TYPE "LBP_typeModeGroup"
TITLE = Mode group signals / Señales de grupo de modos de operación / Betriebsartengruppe Signale
// User data type for block LBP_ModeGroup [DB11] / Tipo de dato de usuario para bloque LBP_ModeGroup [DB11] / Anwender-Datentyp für Baustein LBP_ModeGroup [DB11]
// stored: IsFailsafeCompliant false
   STRUCT
      A_AUTO : Bool;   // Betriebsart AUTOMATIC / Operating mode AUTOMATIC / Modo de operación AUTOMÁTICO
      A_MDA : Bool;   // Betriebsart MDA / Operating mode MDA / Modo de operación MDA
      A_JOG : Bool;   // Betriebsart JOG / Operating mode JOG / Modo de operación JOG
      f0_3 : Bool;
      A_MCDisable : Bool;   // Betriebsartenwechsel deaktivieren / Mode change disable / Desactivar cambio de modo de operación
      A_MGStop : Bool;   // Betriebsartengruppe Stopp / Mode group stop / Parada de grupo de modos de operación
      A_MGStopASp : Bool;   // Betriebsartengruppe Stopp Achsen plus Spindel / Mode group stop axes plus spindle / Parada de grupo de modos de operación ejes y cabezal
      A_MGReset : Bool;   // Betriebsartengruppe Reset / Mode group reset / Reset de grupo de modos de operación
      A_TEACHIN : Bool;   // Maschinenfunktion TEACH IN / Machine function TEACH IN / Función de máquina TEACH IN
      A_REPOS : Bool;   // Maschinenfunktion REPOS / Machine function REPOS / Función de máquina REPOS
      A_REF : Bool;   // Maschinenfunktion REF / Machine function REF / Función de máquina REF
      f1_3 : Bool;
      f1_4 : Bool;
      f1_5 : Bool;
      A_SingleBlock_B : Bool;   // Einzelsatz Typ B / Single block type B / Secuencia individual tipo B
      A_SingleBlock_A : Bool;   // Einzelsatz Typ A / Single block type A / Secuencia individual tipo A
      A_INC1 : Bool;   // INC1
      A_INC10 : Bool;   // INC10
      A_INC100 : Bool;   // INC100
      A_INC1000 : Bool;   // INC1000
      A_INC10000 : Bool;   // INC10000
      A_INCVar : Bool;   // INC-Variable / INC variable / Variable INC
      A_ContManTravel : Bool;   // Kontinuierliches Verfahren von Hand / Continuous manual travel / Desplazamiento continuo a mano
      f2_7 : Bool;
      f3 : Byte;
      E_MMC_AUTO : Bool;   // HMI Betriebsart Strobe AUTOMATIC / HMI mode strobe AUTOMATIC / Modo de operación HMI strobe AUTOMÁTICO
      E_MMC_MDA : Bool;   // HMI Betriebsart Strobe MDA / HMI mode strobe MDA / Modo de operación HMI strobe MDA
      E_MMC_JOG : Bool;   // HMI Betriebsart Strobe JOG / HMI mode strobe JOG / Modo de operación HMI strobe JOG
      f4_3 : Bool;
      f4_4 : Bool;
      f4_5 : Bool;
      f4_6 : Bool;
      f4_7 : Bool;
      E_MMC_TEACHIN : Bool;   // HMI Maschinenfunktion Strobe TEACH IN / HMI machine function strobe TEACH IN / Función de máquina HMI strobe TEACH IN
      E_MMC_REPOS : Bool;   // HMI Maschinenfunktion Strobe REPOS / HMI machine function strobe REPOS / Función de máquina HMI strobe REPOS
      E_MMC_REF : Bool;   // HMI Maschinenfunktion Strobe REF / HMI machine function strobe REF / Función de máquina HMI strobe REF
      f5_3 : Bool;
      f5_4 : Bool;
      f5_5 : Bool;
      f5_6 : Bool;
      f5_7 : Bool;
      E_AUTO : Bool;   // Aktive Betriebsart AUTOMATIC / Active operating mode AUTOMATIC / Modo de operación activo AUTOMÁTICO
      E_MDA : Bool;   // Aktive Betriebsart MDA / Active operating mode MDA / Modo de operación activo MDA
      E_JOG : Bool;   // Aktive Betriebsart JOG / Active operating mode JOG / Modo de operación activo JOG
      E_MGOK : Bool;   // Betriebsartengruppe bereit / Mode group ready / Grupo de modos de operación listo
      E_MGreseted : Bool;   // Betriebsartengruppe Reset durchgeführt / Mode group reset performed / Reset de grupo de modos de operación realizado
      E_NCKintJOG : Bool;   // NCK interner JOG aktiv / NCK internal JOG active / NCK JOG interno activo
      f6_6 : Bool;
      E_ChanReset : Bool;   // Alle Kanäle in Reset-Mode / All channels in reset state / Todos los canales en modo Reset
      E_TEACHIN : Bool;   // Aktive Maschinenfunktion TEACH IN / Active machine function TEACH IN / Función de máquina activa TEACH IN
      E_REPOS : Bool;   // Aktive Maschinenfunktion REPOS / Active machine function REPOS / Función de máquina activa REPOS
      E_REF : Bool;   // Aktive Maschinenfunktion REF / Active machine function REF / Función de máquina activa REF
      f7_3 : Bool;
      f7_4 : Bool;
      f7_5 : Bool;
      f7_6 : Bool;
      f7_7 : Bool;
      E_INC1 : Bool;   // INC1
      E_INC10 : Bool;   // INC10
      E_INC100 : Bool;   // INC100
      E_INC1000 : Bool;   // INC1000
      E_INC10000 : Bool;   // INC10000
      E_INCVar : Bool;   // INC-Variable / INC variable / Variable INC
      E_ContManTravelAct : Bool;   // Kontinuierliches manuelles Verfahren aktiv / Continuous manual travel active / Desplazamiento manual continuo activo
      f8_7 : Bool;
      f9 : Byte;
      E_HMI_INC1 : Bool;   // INC1 vom HMI / INC1 from HMI / INC1 de HMI
      E_HMI_INC10 : Bool;   // INC10 vom HMI / INC10 from HMI / INC10 de HMI
      E_HMI_INC100 : Bool;   // INC100 vom HMI / INC100 from HMI / INC100 de HMI
      E_HMI_INC1000 : Bool;   // INC1000 vom HMI / INC1000 from HMI / INC1000 de HMI
      E_HMI_INC10000 : Bool;   // INC10000 vom HMI / INC10000 from HMI / INC10000 de HMI
      E_HMI_INCVar : Bool;   // INC-Variable vom HMI / INC variable from HMI / Variable INC de HMI
      E_HMI_ContManTravel : Bool;   // Kontinuierliches manuelles Verfahren vom HMI aktiv / Continuous manual travel active from HMI / Desplazamiento manual continuo activo desde HMI
      f10_7 : Bool;
      f11 : Byte;
      f12 : Array[12..19] of Byte;
      MG : Array[2..10] of Struct   // Nächste Betriebsartengruppe vom DBB20, wie bisher / next mode group from DBB20, as before / Próximo grupo de modos de operación del DBB20 como hasta ahora
         A_AUTO : Bool;   // Betriebsart AUTOMATIC / Operating mode AUTOMATIC / Modo de operación AUTOMÁTICO
         A_MDA : Bool;   // Betriebsart MDA / Operating mode MDA / Modo de operación MDA
         A_JOG : Bool;   // Betriebsart JOG / Operating mode JOG / Modo de operación JOG
         f0_3 : Bool;
         A_MCDisable : Bool;   // Betriebsartenwechsel deaktivieren / Mode change disable / Desactivar cambio de modo de operación
         A_MGStop : Bool;   // Betriebsartengruppe Stopp / Mode group stop / Parada de grupo de modos de operación
         A_MGStopASp : Bool;   // Betriebsartengruppe Stopp Achsen plus Spindel / Mode group stop axes plus spindle / Parada de grupo de modos de operación ejes y cabezal
         A_MGReset : Bool;   // Betriebsartengruppe Reset / Mode group reset / Reset de grupo de modos de operación
         A_TEACHIN : Bool;   // Maschinenfunktion TEACH IN / Machine function TEACH IN / Función de máquina TEACH IN
         A_REPOS : Bool;   // Maschinenfunktion REPOS / Machine function REPOS / Función de máquina REPOS
         A_REF : Bool;   // Maschinenfunktion REF / Machine function REF / Función de máquina REF
         f1_3 : Bool;
         f1_4 : Bool;
         f1_5 : Bool;
         A_SingleBlock_B : Bool;   // Einzelsatz Typ B / Single block type B / Secuencia individual tipo B
         A_SingleBlock_A : Bool;   // Einzelsatz Typ A / Single block type A / Secuencia individual tipo A
         A_INC1 : Bool;   // INC1
         A_INC10 : Bool;   // INC10
         A_INC100 : Bool;   // INC100
         A_INC1000 : Bool;   // INC1000
         A_INC10000 : Bool;   // INC10000
         A_INCVar : Bool;   // INC-Variable / INC variable / Variable INC
         A_ContManTravel : Bool;   // Kontinuierliches Verfahren von Hand / Continuous manual travel / Desplazamiento continuo a mano
         f2_7 : Bool;
         f3 : Byte;
         E_MMC_AUTO : Bool;   // HMI Betriebsart Strobe AUTOMATIC / HMI mode strobe AUTOMATIC / Modo de operación HMI strobe AUTOMÁTICO
         E_MMC_MDA : Bool;   // HMI Betriebsart Strobe MDA / HMI mode strobe MDA / Modo de operación HMI strobe MDA
         E_MMC_JOG : Bool;   // HMI Betriebsart Strobe JOG / HMI mode strobe JOG / Modo de operación HMI strobe JOG
         f4_3 : Bool;
         f4_4 : Bool;
         f4_5 : Bool;
         f4_6 : Bool;
         f4_7 : Bool;
         E_MMC_TEACHIN : Bool;   // HMI Maschinenfunktion Strobe TEACH IN / HMI machine function strobe TEACH IN / Función de máquina HMI strobe TEACH IN
         E_MMC_REPOS : Bool;   // HMI Maschinenfunktion Strobe REPOS / HMI machine function strobe REPOS / Función de máquina HMI strobe REPOS
         E_MMC_REF : Bool;   // HMI Maschinenfunktion Strobe REF / HMI machine function strobe REF / Función de máquina HMI strobe REF
         f5_3 : Bool;
         f5_4 : Bool;
         f5_5 : Bool;
         f5_6 : Bool;
         f5_7 : Bool;
         E_AUTO : Bool;   // Aktive Betriebsart AUTOMATIC / Active operating mode AUTOMATIC / Modo de operación activo AUTOMÁTICO
         E_MDA : Bool;   // Aktive Betriebsart MDA / Active operating mode MDA / Modo de operación activo MDA
         E_JOG : Bool;   // Aktive Betriebsart JOG / Active operating mode JOG / Modo de operación activo JOG
         E_MGOK : Bool;   // Betriebsartengruppe bereit / Mode group ready / Grupo de modos de operación listo
         E_MGreseted : Bool;   // Betriebsartengruppe Reset / Mode group reset / Reset de grupo de modos de operación
         E_NCKintJOG : Bool;   // NCK interner JOG aktiv / NCK internal JOG active / NCK JOG interno activo
         f6_6 : Bool;
         E_ChanReset : Bool;   // Alle Kanäle in Reset-Mode / All channels in reset state / Todos los canales en modo Reset
         E_TEACHIN : Bool;   // Aktive Maschinenfunktion TEACH IN / Active machine function TEACH IN / Función de máquina activa TEACH IN
         E_REPOS : Bool;   // Aktive Maschinenfunktion REPOS / Active machine function REPOS / Función de máquina activa REPOS
         E_REF : Bool;   // Aktive Maschinenfunktion REF / Active machine function REF / Función de máquina activa REF
         f7_3 : Bool;
         f7_4 : Bool;
         f7_5 : Bool;
         f7_6 : Bool;
         f7_7 : Bool;
         E_INC1 : Bool;   // INC1
         E_INC10 : Bool;   // INC10
         E_INC100 : Bool;   // INC100
         E_INC1000 : Bool;   // INC1000
         E_INC10000 : Bool;   // INC10000
         E_INCVar : Bool;   // INC-Variable / INC variable / Variable INC
         E_ContManTravelAct : Bool;   // Kontinuierliches manuelles Verfahren aktiv / Continuous manual travel active / Desplazamiento manual continuo activo
         f8_7 : Bool;
         f9 : Byte;
         E_HMI_INC1 : Bool;   // INC1 vom HMI / INC1 from HMI / INC1 de HMI
         E_HMI_INC10 : Bool;   // INC10 vom HMI / INC10 from HMI / INC10 de HMI
         E_HMI_INC100 : Bool;   // INC100 vom HMI / INC100 from HMI / INC100 de HMI
         E_HMI_INC1000 : Bool;   // INC1000 vom HMI / INC1000 from HMI / INC1000 de HMI
         E_HMI_INC10000 : Bool;   // INC10000 vom HMI / INC10000 from HMI / INC10000 de HMI
         E_HMI_INCVar : Bool;   // INC-Variable vom HMI / INC variable from HMI / Variable INC de HMI
         E_HMI_ContManTravel : Bool;   // Kontinuierliches manuelles Verfahren vom HMI aktiv / Continuous manual travel active from HMI / Desplazamiento manual continuo activo desde HMI
         f10_7 : Bool;
         f11 : Byte;
         f12 : Array[12..19] of Byte;
      END_STRUCT;
   END_STRUCT;
   // // MG[3].A_AUTO : Betriebsart AUTOMATIC / Operating mode AUTOMATIC / Modo de operación AUTOMÁTICO
   // // MG[4].A_AUTO : Betriebsart AUTOMATIC / Operating mode AUTOMATIC / Modo de operación AUTOMÁTICO
   // // MG[5].A_AUTO : Betriebsart AUTOMATIC / Operating mode AUTOMATIC / Modo de operación AUTOMÁTICO
   // // MG[6].A_AUTO : Betriebsart AUTOMATIC / Operating mode AUTOMATIC / Modo de operación AUTOMÁTICO
   // // MG[7].A_AUTO : Betriebsart AUTOMATIC / Operating mode AUTOMATIC / Modo de operación AUTOMÁTICO
   // // MG[8].A_AUTO : Betriebsart AUTOMATIC / Operating mode AUTOMATIC / Modo de operación AUTOMÁTICO
   // // MG[9].A_AUTO : Betriebsart AUTOMATIC / Operating mode AUTOMATIC / Modo de operación AUTOMÁTICO
   // // MG[10].A_AUTO : Betriebsart AUTOMATIC / Operating mode AUTOMATIC / Modo de operación AUTOMÁTICO
   // // MG[3].A_MDA : Betriebsart MDA / Operating mode MDA / Modo de operación MDA
   // // MG[4].A_MDA : Betriebsart MDA / Operating mode MDA / Modo de operación MDA
   // // MG[5].A_MDA : Betriebsart MDA / Operating mode MDA / Modo de operación MDA
   // // MG[6].A_MDA : Betriebsart MDA / Operating mode MDA / Modo de operación MDA
   // // MG[7].A_MDA : Betriebsart MDA / Operating mode MDA / Modo de operación MDA
   // // MG[8].A_MDA : Betriebsart MDA / Operating mode MDA / Modo de operación MDA
   // // MG[9].A_MDA : Betriebsart MDA / Operating mode MDA / Modo de operación MDA
   // // MG[10].A_MDA : Betriebsart MDA / Operating mode MDA / Modo de operación MDA
   // // MG[3].A_JOG : Betriebsart JOG / Operating mode JOG / Modo de operación JOG
   // // MG[4].A_JOG : Betriebsart JOG / Operating mode JOG / Modo de operación JOG
   // // MG[5].A_JOG : Betriebsart JOG / Operating mode JOG / Modo de operación JOG
   // // MG[6].A_JOG : Betriebsart JOG / Operating mode JOG / Modo de operación JOG
   // // MG[7].A_JOG : Betriebsart JOG / Operating mode JOG / Modo de operación JOG
   // // MG[8].A_JOG : Betriebsart JOG / Operating mode JOG / Modo de operación JOG
   // // MG[9].A_JOG : Betriebsart JOG / Operating mode JOG / Modo de operación JOG
   // // MG[10].A_JOG : Betriebsart JOG / Operating mode JOG / Modo de operación JOG
   // // MG[3].A_MCDisable : Betriebsartenwechsel deaktivieren / Mode change disable / Desactivar cambio de modo de operación
   // // MG[4].A_MCDisable : Betriebsartenwechsel deaktivieren / Mode change disable / Desactivar cambio de modo de operación
   // // MG[5].A_MCDisable : Betriebsartenwechsel deaktivieren / Mode change disable / Desactivar cambio de modo de operación
   // // MG[6].A_MCDisable : Betriebsartenwechsel deaktivieren / Mode change disable / Desactivar cambio de modo de operación
   // // MG[7].A_MCDisable : Betriebsartenwechsel deaktivieren / Mode change disable / Desactivar cambio de modo de operación
   // // MG[8].A_MCDisable : Betriebsartenwechsel deaktivieren / Mode change disable / Desactivar cambio de modo de operación
   // // MG[9].A_MCDisable : Betriebsartenwechsel deaktivieren / Mode change disable / Desactivar cambio de modo de operación
   // // MG[10].A_MCDisable : Betriebsartenwechsel deaktivieren / Mode change disable / Desactivar cambio de modo de operación
   // // MG[3].A_MGStop : Betriebsartengruppe Stopp / Mode group stop / Parada de grupo de modos de operación
   // // MG[4].A_MGStop : Betriebsartengruppe Stopp / Mode group stop / Parada de grupo de modos de operación
   // // MG[5].A_MGStop : Betriebsartengruppe Stopp / Mode group stop / Parada de grupo de modos de operación
   // // MG[6].A_MGStop : Betriebsartengruppe Stopp / Mode group stop / Parada de grupo de modos de operación
   // // MG[7].A_MGStop : Betriebsartengruppe Stopp / Mode group stop / Parada de grupo de modos de operación
   // // MG[8].A_MGStop : Betriebsartengruppe Stopp / Mode group stop / Parada de grupo de modos de operación
   // // MG[9].A_MGStop : Betriebsartengruppe Stopp / Mode group stop / Parada de grupo de modos de operación
   // // MG[10].A_MGStop : Betriebsartengruppe Stopp / Mode group stop / Parada de grupo de modos de operación
   // // MG[3].A_MGStopASp : Betriebsartengruppe Stopp Achsen plus Spindel / Mode group stop axes plus spindle / Parada de grupo de modos de operación ejes y cabezal
   // // MG[4].A_MGStopASp : Betriebsartengruppe Stopp Achsen plus Spindel / Mode group stop axes plus spindle / Parada de grupo de modos de operación ejes y cabezal
   // // MG[5].A_MGStopASp : Betriebsartengruppe Stopp Achsen plus Spindel / Mode group stop axes plus spindle / Parada de grupo de modos de operación ejes y cabezal
   // // MG[6].A_MGStopASp : Betriebsartengruppe Stopp Achsen plus Spindel / Mode group stop axes plus spindle / Parada de grupo de modos de operación ejes y cabezal
   // // MG[7].A_MGStopASp : Betriebsartengruppe Stopp Achsen plus Spindel / Mode group stop axes plus spindle / Parada de grupo de modos de operación ejes y cabezal
   // // MG[8].A_MGStopASp : Betriebsartengruppe Stopp Achsen plus Spindel / Mode group stop axes plus spindle / Parada de grupo de modos de operación ejes y cabezal
   // // MG[9].A_MGStopASp : Betriebsartengruppe Stopp Achsen plus Spindel / Mode group stop axes plus spindle / Parada de grupo de modos de operación ejes y cabezal
   // // MG[10].A_MGStopASp : Betriebsartengruppe Stopp Achsen plus Spindel / Mode group stop axes plus spindle / Parada de grupo de modos de operación ejes y cabezal
   // // MG[3].A_MGReset : Betriebsartengruppe Reset / Mode group reset / Reset de grupo de modos de operación
   // // MG[4].A_MGReset : Betriebsartengruppe Reset / Mode group reset / Reset de grupo de modos de operación
   // // MG[5].A_MGReset : Betriebsartengruppe Reset / Mode group reset / Reset de grupo de modos de operación
   // // MG[6].A_MGReset : Betriebsartengruppe Reset / Mode group reset / Reset de grupo de modos de operación
   // // MG[7].A_MGReset : Betriebsartengruppe Reset / Mode group reset / Reset de grupo de modos de operación
   // // MG[8].A_MGReset : Betriebsartengruppe Reset / Mode group reset / Reset de grupo de modos de operación
   // // MG[9].A_MGReset : Betriebsartengruppe Reset / Mode group reset / Reset de grupo de modos de operación
   // // MG[10].A_MGReset : Betriebsartengruppe Reset / Mode group reset / Reset de grupo de modos de operación
   // // MG[3].A_TEACHIN : Maschinenfunktion TEACH IN / Machine function TEACH IN / Función de máquina TEACH IN
   // // MG[4].A_TEACHIN : Maschinenfunktion TEACH IN / Machine function TEACH IN / Función de máquina TEACH IN
   // // MG[5].A_TEACHIN : Maschinenfunktion TEACH IN / Machine function TEACH IN / Función de máquina TEACH IN
   // // MG[6].A_TEACHIN : Maschinenfunktion TEACH IN / Machine function TEACH IN / Función de máquina TEACH IN
   // // MG[7].A_TEACHIN : Maschinenfunktion TEACH IN / Machine function TEACH IN / Función de máquina TEACH IN
   // // MG[8].A_TEACHIN : Maschinenfunktion TEACH IN / Machine function TEACH IN / Función de máquina TEACH IN
   // // MG[9].A_TEACHIN : Maschinenfunktion TEACH IN / Machine function TEACH IN / Función de máquina TEACH IN
   // // MG[10].A_TEACHIN : Maschinenfunktion TEACH IN / Machine function TEACH IN / Función de máquina TEACH IN
   // // MG[3].A_REPOS : Maschinenfunktion REPOS / Machine function REPOS / Función de máquina REPOS
   // // MG[4].A_REPOS : Maschinenfunktion REPOS / Machine function REPOS / Función de máquina REPOS
   // // MG[5].A_REPOS : Maschinenfunktion REPOS / Machine function REPOS / Función de máquina REPOS
   // // MG[6].A_REPOS : Maschinenfunktion REPOS / Machine function REPOS / Función de máquina REPOS
   // // MG[7].A_REPOS : Maschinenfunktion REPOS / Machine function REPOS / Función de máquina REPOS
   // // MG[8].A_REPOS : Maschinenfunktion REPOS / Machine function REPOS / Función de máquina REPOS
   // // MG[9].A_REPOS : Maschinenfunktion REPOS / Machine function REPOS / Función de máquina REPOS
   // // MG[10].A_REPOS : Maschinenfunktion REPOS / Machine function REPOS / Función de máquina REPOS
   // // MG[3].A_REF : Maschinenfunktion REF / Machine function REF / Función de máquina REF
   // // MG[4].A_REF : Maschinenfunktion REF / Machine function REF / Función de máquina REF
   // // MG[5].A_REF : Maschinenfunktion REF / Machine function REF / Función de máquina REF
   // // MG[6].A_REF : Maschinenfunktion REF / Machine function REF / Función de máquina REF
   // // MG[7].A_REF : Maschinenfunktion REF / Machine function REF / Función de máquina REF
   // // MG[8].A_REF : Maschinenfunktion REF / Machine function REF / Función de máquina REF
   // // MG[9].A_REF : Maschinenfunktion REF / Machine function REF / Función de máquina REF
   // // MG[10].A_REF : Maschinenfunktion REF / Machine function REF / Función de máquina REF
   // // MG[3].A_SingleBlock_B : Einzelsatz Typ B / Single block type B / Secuencia individual tipo B
   // // MG[4].A_SingleBlock_B : Einzelsatz Typ B / Single block type B / Secuencia individual tipo B
   // // MG[5].A_SingleBlock_B : Einzelsatz Typ B / Single block type B / Secuencia individual tipo B
   // // MG[6].A_SingleBlock_B : Einzelsatz Typ B / Single block type B / Secuencia individual tipo B
   // // MG[7].A_SingleBlock_B : Einzelsatz Typ B / Single block type B / Secuencia individual tipo B
   // // MG[8].A_SingleBlock_B : Einzelsatz Typ B / Single block type B / Secuencia individual tipo B
   // // MG[9].A_SingleBlock_B : Einzelsatz Typ B / Single block type B / Secuencia individual tipo B
   // // MG[10].A_SingleBlock_B : Einzelsatz Typ B / Single block type B / Secuencia individual tipo B
   // // MG[3].A_SingleBlock_A : Einzelsatz Typ A / Single block type A / Secuencia individual tipo A
   // // MG[4].A_SingleBlock_A : Einzelsatz Typ A / Single block type A / Secuencia individual tipo A
   // // MG[5].A_SingleBlock_A : Einzelsatz Typ A / Single block type A / Secuencia individual tipo A
   // // MG[6].A_SingleBlock_A : Einzelsatz Typ A / Single block type A / Secuencia individual tipo A
   // // MG[7].A_SingleBlock_A : Einzelsatz Typ A / Single block type A / Secuencia individual tipo A
   // // MG[8].A_SingleBlock_A : Einzelsatz Typ A / Single block type A / Secuencia individual tipo A
   // // MG[9].A_SingleBlock_A : Einzelsatz Typ A / Single block type A / Secuencia individual tipo A
   // // MG[10].A_SingleBlock_A : Einzelsatz Typ A / Single block type A / Secuencia individual tipo A
   // // MG[3].A_INC1 : INC1
   // // MG[4].A_INC1 : INC1
   // // MG[5].A_INC1 : INC1
   // // MG[6].A_INC1 : INC1
   // // MG[7].A_INC1 : INC1
   // // MG[8].A_INC1 : INC1
   // // MG[9].A_INC1 : INC1
   // // MG[10].A_INC1 : INC1
   // // MG[3].A_INC10 : INC10
   // // MG[4].A_INC10 : INC10
   // // MG[5].A_INC10 : INC10
   // // MG[6].A_INC10 : INC10
   // // MG[7].A_INC10 : INC10
   // // MG[8].A_INC10 : INC10
   // // MG[9].A_INC10 : INC10
   // // MG[10].A_INC10 : INC10
   // // MG[3].A_INC100 : INC100
   // // MG[4].A_INC100 : INC100
   // // MG[5].A_INC100 : INC100
   // // MG[6].A_INC100 : INC100
   // // MG[7].A_INC100 : INC100
   // // MG[8].A_INC100 : INC100
   // // MG[9].A_INC100 : INC100
   // // MG[10].A_INC100 : INC100
   // // MG[3].A_INC1000 : INC1000
   // // MG[4].A_INC1000 : INC1000
   // // MG[5].A_INC1000 : INC1000
   // // MG[6].A_INC1000 : INC1000
   // // MG[7].A_INC1000 : INC1000
   // // MG[8].A_INC1000 : INC1000
   // // MG[9].A_INC1000 : INC1000
   // // MG[10].A_INC1000 : INC1000
   // // MG[3].A_INC10000 : INC10000
   // // MG[4].A_INC10000 : INC10000
   // // MG[5].A_INC10000 : INC10000
   // // MG[6].A_INC10000 : INC10000
   // // MG[7].A_INC10000 : INC10000
   // // MG[8].A_INC10000 : INC10000
   // // MG[9].A_INC10000 : INC10000
   // // MG[10].A_INC10000 : INC10000
   // // MG[3].A_INCVar : INC-Variable / INC variable / Variable INC
   // // MG[4].A_INCVar : INC-Variable / INC variable / Variable INC
   // // MG[5].A_INCVar : INC-Variable / INC variable / Variable INC
   // // MG[6].A_INCVar : INC-Variable / INC variable / Variable INC
   // // MG[7].A_INCVar : INC-Variable / INC variable / Variable INC
   // // MG[8].A_INCVar : INC-Variable / INC variable / Variable INC
   // // MG[9].A_INCVar : INC-Variable / INC variable / Variable INC
   // // MG[10].A_INCVar : INC-Variable / INC variable / Variable INC
   // // MG[3].A_ContManTravel : Kontinuierliches Verfahren von Hand / Continuous manual travel / Desplazamiento continuo a mano
   // // MG[4].A_ContManTravel : Kontinuierliches Verfahren von Hand / Continuous manual travel / Desplazamiento continuo a mano
   // // MG[5].A_ContManTravel : Kontinuierliches Verfahren von Hand / Continuous manual travel / Desplazamiento continuo a mano
   // // MG[6].A_ContManTravel : Kontinuierliches Verfahren von Hand / Continuous manual travel / Desplazamiento continuo a mano
   // // MG[7].A_ContManTravel : Kontinuierliches Verfahren von Hand / Continuous manual travel / Desplazamiento continuo a mano
   // // MG[8].A_ContManTravel : Kontinuierliches Verfahren von Hand / Continuous manual travel / Desplazamiento continuo a mano
   // // MG[9].A_ContManTravel : Kontinuierliches Verfahren von Hand / Continuous manual travel / Desplazamiento continuo a mano
   // // MG[10].A_ContManTravel : Kontinuierliches Verfahren von Hand / Continuous manual travel / Desplazamiento continuo a mano
   // // MG[3].E_MMC_AUTO : HMI Betriebsart Strobe AUTOMATIC / HMI mode strobe AUTOMATIC / Modo de operación HMI strobe AUTOMÁTICO
   // // MG[4].E_MMC_AUTO : HMI Betriebsart Strobe AUTOMATIC / HMI mode strobe AUTOMATIC / Modo de operación HMI strobe AUTOMÁTICO
   // // MG[5].E_MMC_AUTO : HMI Betriebsart Strobe AUTOMATIC / HMI mode strobe AUTOMATIC / Modo de operación HMI strobe AUTOMÁTICO
   // // MG[6].E_MMC_AUTO : HMI Betriebsart Strobe AUTOMATIC / HMI mode strobe AUTOMATIC / Modo de operación HMI strobe AUTOMÁTICO
   // // MG[7].E_MMC_AUTO : HMI Betriebsart Strobe AUTOMATIC / HMI mode strobe AUTOMATIC / Modo de operación HMI strobe AUTOMÁTICO
   // // MG[8].E_MMC_AUTO : HMI Betriebsart Strobe AUTOMATIC / HMI mode strobe AUTOMATIC / Modo de operación HMI strobe AUTOMÁTICO
   // // MG[9].E_MMC_AUTO : HMI Betriebsart Strobe AUTOMATIC / HMI mode strobe AUTOMATIC / Modo de operación HMI strobe AUTOMÁTICO
   // // MG[10].E_MMC_AUTO : HMI Betriebsart Strobe AUTOMATIC / HMI mode strobe AUTOMATIC / Modo de operación HMI strobe AUTOMÁTICO
   // // MG[3].E_MMC_MDA : HMI Betriebsart Strobe MDA / HMI mode strobe MDA / Modo de operación HMI strobe MDA
   // // MG[4].E_MMC_MDA : HMI Betriebsart Strobe MDA / HMI mode strobe MDA / Modo de operación HMI strobe MDA
   // // MG[5].E_MMC_MDA : HMI Betriebsart Strobe MDA / HMI mode strobe MDA / Modo de operación HMI strobe MDA
   // // MG[6].E_MMC_MDA : HMI Betriebsart Strobe MDA / HMI mode strobe MDA / Modo de operación HMI strobe MDA
   // // MG[7].E_MMC_MDA : HMI Betriebsart Strobe MDA / HMI mode strobe MDA / Modo de operación HMI strobe MDA
   // // MG[8].E_MMC_MDA : HMI Betriebsart Strobe MDA / HMI mode strobe MDA / Modo de operación HMI strobe MDA
   // // MG[9].E_MMC_MDA : HMI Betriebsart Strobe MDA / HMI mode strobe MDA / Modo de operación HMI strobe MDA
   // // MG[10].E_MMC_MDA : HMI Betriebsart Strobe MDA / HMI mode strobe MDA / Modo de operación HMI strobe MDA
   // // MG[3].E_MMC_JOG : HMI Betriebsart Strobe JOG / HMI mode strobe JOG / Modo de operación HMI strobe JOG
   // // MG[4].E_MMC_JOG : HMI Betriebsart Strobe JOG / HMI mode strobe JOG / Modo de operación HMI strobe JOG
   // // MG[5].E_MMC_JOG : HMI Betriebsart Strobe JOG / HMI mode strobe JOG / Modo de operación HMI strobe JOG
   // // MG[6].E_MMC_JOG : HMI Betriebsart Strobe JOG / HMI mode strobe JOG / Modo de operación HMI strobe JOG
   // // MG[7].E_MMC_JOG : HMI Betriebsart Strobe JOG / HMI mode strobe JOG / Modo de operación HMI strobe JOG
   // // MG[8].E_MMC_JOG : HMI Betriebsart Strobe JOG / HMI mode strobe JOG / Modo de operación HMI strobe JOG
   // // MG[9].E_MMC_JOG : HMI Betriebsart Strobe JOG / HMI mode strobe JOG / Modo de operación HMI strobe JOG
   // // MG[10].E_MMC_JOG : HMI Betriebsart Strobe JOG / HMI mode strobe JOG / Modo de operación HMI strobe JOG
   // // MG[3].E_MMC_TEACHIN : HMI Maschinenfunktion Strobe TEACH IN / HMI machine function strobe TEACH IN / Función de máquina HMI strobe TEACH IN
   // // MG[4].E_MMC_TEACHIN : HMI Maschinenfunktion Strobe TEACH IN / HMI machine function strobe TEACH IN / Función de máquina HMI strobe TEACH IN
   // // MG[5].E_MMC_TEACHIN : HMI Maschinenfunktion Strobe TEACH IN / HMI machine function strobe TEACH IN / Función de máquina HMI strobe TEACH IN
   // // MG[6].E_MMC_TEACHIN : HMI Maschinenfunktion Strobe TEACH IN / HMI machine function strobe TEACH IN / Función de máquina HMI strobe TEACH IN
   // // MG[7].E_MMC_TEACHIN : HMI Maschinenfunktion Strobe TEACH IN / HMI machine function strobe TEACH IN / Función de máquina HMI strobe TEACH IN
   // // MG[8].E_MMC_TEACHIN : HMI Maschinenfunktion Strobe TEACH IN / HMI machine function strobe TEACH IN / Función de máquina HMI strobe TEACH IN
   // // MG[9].E_MMC_TEACHIN : HMI Maschinenfunktion Strobe TEACH IN / HMI machine function strobe TEACH IN / Función de máquina HMI strobe TEACH IN
   // // MG[10].E_MMC_TEACHIN : HMI Maschinenfunktion Strobe TEACH IN / HMI machine function strobe TEACH IN / Función de máquina HMI strobe TEACH IN
   // // MG[3].E_MMC_REPOS : HMI Maschinenfunktion Strobe REPOS / HMI machine function strobe REPOS / Función de máquina HMI strobe REPOS
   // // MG[4].E_MMC_REPOS : HMI Maschinenfunktion Strobe REPOS / HMI machine function strobe REPOS / Función de máquina HMI strobe REPOS
   // // MG[5].E_MMC_REPOS : HMI Maschinenfunktion Strobe REPOS / HMI machine function strobe REPOS / Función de máquina HMI strobe REPOS
   // // MG[6].E_MMC_REPOS : HMI Maschinenfunktion Strobe REPOS / HMI machine function strobe REPOS / Función de máquina HMI strobe REPOS
   // // MG[7].E_MMC_REPOS : HMI Maschinenfunktion Strobe REPOS / HMI machine function strobe REPOS / Función de máquina HMI strobe REPOS
   // // MG[8].E_MMC_REPOS : HMI Maschinenfunktion Strobe REPOS / HMI machine function strobe REPOS / Función de máquina HMI strobe REPOS
   // // MG[9].E_MMC_REPOS : HMI Maschinenfunktion Strobe REPOS / HMI machine function strobe REPOS / Función de máquina HMI strobe REPOS
   // // MG[10].E_MMC_REPOS : HMI Maschinenfunktion Strobe REPOS / HMI machine function strobe REPOS / Función de máquina HMI strobe REPOS
   // // MG[3].E_MMC_REF : HMI Maschinenfunktion Strobe REF / HMI machine function strobe REF / Función de máquina HMI strobe REF
   // // MG[4].E_MMC_REF : HMI Maschinenfunktion Strobe REF / HMI machine function strobe REF / Función de máquina HMI strobe REF
   // // MG[5].E_MMC_REF : HMI Maschinenfunktion Strobe REF / HMI machine function strobe REF / Función de máquina HMI strobe REF
   // // MG[6].E_MMC_REF : HMI Maschinenfunktion Strobe REF / HMI machine function strobe REF / Función de máquina HMI strobe REF
   // // MG[7].E_MMC_REF : HMI Maschinenfunktion Strobe REF / HMI machine function strobe REF / Función de máquina HMI strobe REF
   // // MG[8].E_MMC_REF : HMI Maschinenfunktion Strobe REF / HMI machine function strobe REF / Función de máquina HMI strobe REF
   // // MG[9].E_MMC_REF : HMI Maschinenfunktion Strobe REF / HMI machine function strobe REF / Función de máquina HMI strobe REF
   // // MG[10].E_MMC_REF : HMI Maschinenfunktion Strobe REF / HMI machine function strobe REF / Función de máquina HMI strobe REF
   // // MG[3].E_AUTO : Aktive Betriebsart AUTOMATIC / Active operating mode AUTOMATIC / Modo de operación activo AUTOMÁTICO
   // // MG[4].E_AUTO : Aktive Betriebsart AUTOMATIC / Active operating mode AUTOMATIC / Modo de operación activo AUTOMÁTICO
   // // MG[5].E_AUTO : Aktive Betriebsart AUTOMATIC / Active operating mode AUTOMATIC / Modo de operación activo AUTOMÁTICO
   // // MG[6].E_AUTO : Aktive Betriebsart AUTOMATIC / Active operating mode AUTOMATIC / Modo de operación activo AUTOMÁTICO
   // // MG[7].E_AUTO : Aktive Betriebsart AUTOMATIC / Active operating mode AUTOMATIC / Modo de operación activo AUTOMÁTICO
   // // MG[8].E_AUTO : Aktive Betriebsart AUTOMATIC / Active operating mode AUTOMATIC / Modo de operación activo AUTOMÁTICO
   // // MG[9].E_AUTO : Aktive Betriebsart AUTOMATIC / Active operating mode AUTOMATIC / Modo de operación activo AUTOMÁTICO
   // // MG[10].E_AUTO : Aktive Betriebsart AUTOMATIC / Active operating mode AUTOMATIC / Modo de operación activo AUTOMÁTICO
   // // MG[3].E_MDA : Aktive Betriebsart MDA / Active operating mode MDA / Modo de operación activo MDA
   // // MG[4].E_MDA : Aktive Betriebsart MDA / Active operating mode MDA / Modo de operación activo MDA
   // // MG[5].E_MDA : Aktive Betriebsart MDA / Active operating mode MDA / Modo de operación activo MDA
   // // MG[6].E_MDA : Aktive Betriebsart MDA / Active operating mode MDA / Modo de operación activo MDA
   // // MG[7].E_MDA : Aktive Betriebsart MDA / Active operating mode MDA / Modo de operación activo MDA
   // // MG[8].E_MDA : Aktive Betriebsart MDA / Active operating mode MDA / Modo de operación activo MDA
   // // MG[9].E_MDA : Aktive Betriebsart MDA / Active operating mode MDA / Modo de operación activo MDA
   // // MG[10].E_MDA : Aktive Betriebsart MDA / Active operating mode MDA / Modo de operación activo MDA
   // // MG[3].E_JOG : Aktive Betriebsart JOG / Active operating mode JOG / Modo de operación activo JOG
   // // MG[4].E_JOG : Aktive Betriebsart JOG / Active operating mode JOG / Modo de operación activo JOG
   // // MG[5].E_JOG : Aktive Betriebsart JOG / Active operating mode JOG / Modo de operación activo JOG
   // // MG[6].E_JOG : Aktive Betriebsart JOG / Active operating mode JOG / Modo de operación activo JOG
   // // MG[7].E_JOG : Aktive Betriebsart JOG / Active operating mode JOG / Modo de operación activo JOG
   // // MG[8].E_JOG : Aktive Betriebsart JOG / Active operating mode JOG / Modo de operación activo JOG
   // // MG[9].E_JOG : Aktive Betriebsart JOG / Active operating mode JOG / Modo de operación activo JOG
   // // MG[10].E_JOG : Aktive Betriebsart JOG / Active operating mode JOG / Modo de operación activo JOG
   // // MG[3].E_MGOK : Betriebsartengruppe bereit / Mode group ready / Grupo de modos de operación listo
   // // MG[4].E_MGOK : Betriebsartengruppe bereit / Mode group ready / Grupo de modos de operación listo
   // // MG[5].E_MGOK : Betriebsartengruppe bereit / Mode group ready / Grupo de modos de operación listo
   // // MG[6].E_MGOK : Betriebsartengruppe bereit / Mode group ready / Grupo de modos de operación listo
   // // MG[7].E_MGOK : Betriebsartengruppe bereit / Mode group ready / Grupo de modos de operación listo
   // // MG[8].E_MGOK : Betriebsartengruppe bereit / Mode group ready / Grupo de modos de operación listo
   // // MG[9].E_MGOK : Betriebsartengruppe bereit / Mode group ready / Grupo de modos de operación listo
   // // MG[10].E_MGOK : Betriebsartengruppe bereit / Mode group ready / Grupo de modos de operación listo
   // // MG[3].E_MGreseted : Betriebsartengruppe Reset / Mode group reset / Reset de grupo de modos de operación
   // // MG[4].E_MGreseted : Betriebsartengruppe Reset / Mode group reset / Reset de grupo de modos de operación
   // // MG[5].E_MGreseted : Betriebsartengruppe Reset / Mode group reset / Reset de grupo de modos de operación
   // // MG[6].E_MGreseted : Betriebsartengruppe Reset / Mode group reset / Reset de grupo de modos de operación
   // // MG[7].E_MGreseted : Betriebsartengruppe Reset / Mode group reset / Reset de grupo de modos de operación
   // // MG[8].E_MGreseted : Betriebsartengruppe Reset / Mode group reset / Reset de grupo de modos de operación
   // // MG[9].E_MGreseted : Betriebsartengruppe Reset / Mode group reset / Reset de grupo de modos de operación
   // // MG[10].E_MGreseted : Betriebsartengruppe Reset / Mode group reset / Reset de grupo de modos de operación
   // // MG[3].E_NCKintJOG : NCK interner JOG aktiv / NCK internal JOG active / NCK JOG interno activo
   // // MG[4].E_NCKintJOG : NCK interner JOG aktiv / NCK internal JOG active / NCK JOG interno activo
   // // MG[5].E_NCKintJOG : NCK interner JOG aktiv / NCK internal JOG active / NCK JOG interno activo
   // // MG[6].E_NCKintJOG : NCK interner JOG aktiv / NCK internal JOG active / NCK JOG interno activo
   // // MG[7].E_NCKintJOG : NCK interner JOG aktiv / NCK internal JOG active / NCK JOG interno activo
   // // MG[8].E_NCKintJOG : NCK interner JOG aktiv / NCK internal JOG active / NCK JOG interno activo
   // // MG[9].E_NCKintJOG : NCK interner JOG aktiv / NCK internal JOG active / NCK JOG interno activo
   // // MG[10].E_NCKintJOG : NCK interner JOG aktiv / NCK internal JOG active / NCK JOG interno activo
   // // MG[3].E_ChanReset : Alle Kanäle in Reset-Mode / All channels in reset state / Todos los canales en modo Reset
   // // MG[4].E_ChanReset : Alle Kanäle in Reset-Mode / All channels in reset state / Todos los canales en modo Reset
   // // MG[5].E_ChanReset : Alle Kanäle in Reset-Mode / All channels in reset state / Todos los canales en modo Reset
   // // MG[6].E_ChanReset : Alle Kanäle in Reset-Mode / All channels in reset state / Todos los canales en modo Reset
   // // MG[7].E_ChanReset : Alle Kanäle in Reset-Mode / All channels in reset state / Todos los canales en modo Reset
   // // MG[8].E_ChanReset : Alle Kanäle in Reset-Mode / All channels in reset state / Todos los canales en modo Reset
   // // MG[9].E_ChanReset : Alle Kanäle in Reset-Mode / All channels in reset state / Todos los canales en modo Reset
   // // MG[10].E_ChanReset : Alle Kanäle in Reset-Mode / All channels in reset state / Todos los canales en modo Reset
   // // MG[3].E_TEACHIN : Aktive Maschinenfunktion TEACH IN / Active machine function TEACH IN / Función de máquina activa TEACH IN
   // // MG[4].E_TEACHIN : Aktive Maschinenfunktion TEACH IN / Active machine function TEACH IN / Función de máquina activa TEACH IN
   // // MG[5].E_TEACHIN : Aktive Maschinenfunktion TEACH IN / Active machine function TEACH IN / Función de máquina activa TEACH IN
   // // MG[6].E_TEACHIN : Aktive Maschinenfunktion TEACH IN / Active machine function TEACH IN / Función de máquina activa TEACH IN
   // // MG[7].E_TEACHIN : Aktive Maschinenfunktion TEACH IN / Active machine function TEACH IN / Función de máquina activa TEACH IN
   // // MG[8].E_TEACHIN : Aktive Maschinenfunktion TEACH IN / Active machine function TEACH IN / Función de máquina activa TEACH IN
   // // MG[9].E_TEACHIN : Aktive Maschinenfunktion TEACH IN / Active machine function TEACH IN / Función de máquina activa TEACH IN
   // // MG[10].E_TEACHIN : Aktive Maschinenfunktion TEACH IN / Active machine function TEACH IN / Función de máquina activa TEACH IN
   // // MG[3].E_REPOS : Aktive Maschinenfunktion REPOS / Active machine function REPOS / Función de máquina activa REPOS
   // // MG[4].E_REPOS : Aktive Maschinenfunktion REPOS / Active machine function REPOS / Función de máquina activa REPOS
   // // MG[5].E_REPOS : Aktive Maschinenfunktion REPOS / Active machine function REPOS / Función de máquina activa REPOS
   // // MG[6].E_REPOS : Aktive Maschinenfunktion REPOS / Active machine function REPOS / Función de máquina activa REPOS
   // // MG[7].E_REPOS : Aktive Maschinenfunktion REPOS / Active machine function REPOS / Función de máquina activa REPOS
   // // MG[8].E_REPOS : Aktive Maschinenfunktion REPOS / Active machine function REPOS / Función de máquina activa REPOS
   // // MG[9].E_REPOS : Aktive Maschinenfunktion REPOS / Active machine function REPOS / Función de máquina activa REPOS
   // // MG[10].E_REPOS : Aktive Maschinenfunktion REPOS / Active machine function REPOS / Función de máquina activa REPOS
   // // MG[3].E_REF : Aktive Maschinenfunktion REF / Active machine function REF / Función de máquina activa REF
   // // MG[4].E_REF : Aktive Maschinenfunktion REF / Active machine function REF / Función de máquina activa REF
   // // MG[5].E_REF : Aktive Maschinenfunktion REF / Active machine function REF / Función de máquina activa REF
   // // MG[6].E_REF : Aktive Maschinenfunktion REF / Active machine function REF / Función de máquina activa REF
   // // MG[7].E_REF : Aktive Maschinenfunktion REF / Active machine function REF / Función de máquina activa REF
   // // MG[8].E_REF : Aktive Maschinenfunktion REF / Active machine function REF / Función de máquina activa REF
   // // MG[9].E_REF : Aktive Maschinenfunktion REF / Active machine function REF / Función de máquina activa REF
   // // MG[10].E_REF : Aktive Maschinenfunktion REF / Active machine function REF / Función de máquina activa REF
   // // MG[3].E_INC1 : INC1
   // // MG[4].E_INC1 : INC1
   // // MG[5].E_INC1 : INC1
   // // MG[6].E_INC1 : INC1
   // // MG[7].E_INC1 : INC1
   // // MG[8].E_INC1 : INC1
   // // MG[9].E_INC1 : INC1
   // // MG[10].E_INC1 : INC1
   // // MG[3].E_INC10 : INC10
   // // MG[4].E_INC10 : INC10
   // // MG[5].E_INC10 : INC10
   // // MG[6].E_INC10 : INC10
   // // MG[7].E_INC10 : INC10
   // // MG[8].E_INC10 : INC10
   // // MG[9].E_INC10 : INC10
   // // MG[10].E_INC10 : INC10
   // // MG[3].E_INC100 : INC100
   // // MG[4].E_INC100 : INC100
   // // MG[5].E_INC100 : INC100
   // // MG[6].E_INC100 : INC100
   // // MG[7].E_INC100 : INC100
   // // MG[8].E_INC100 : INC100
   // // MG[9].E_INC100 : INC100
   // // MG[10].E_INC100 : INC100
   // // MG[3].E_INC1000 : INC1000
   // // MG[4].E_INC1000 : INC1000
   // // MG[5].E_INC1000 : INC1000
   // // MG[6].E_INC1000 : INC1000
   // // MG[7].E_INC1000 : INC1000
   // // MG[8].E_INC1000 : INC1000
   // // MG[9].E_INC1000 : INC1000
   // // MG[10].E_INC1000 : INC1000
   // // MG[3].E_INC10000 : INC10000
   // // MG[4].E_INC10000 : INC10000
   // // MG[5].E_INC10000 : INC10000
   // // MG[6].E_INC10000 : INC10000
   // // MG[7].E_INC10000 : INC10000
   // // MG[8].E_INC10000 : INC10000
   // // MG[9].E_INC10000 : INC10000
   // // MG[10].E_INC10000 : INC10000
   // // MG[3].E_INCVar : INC-Variable / INC variable / Variable INC
   // // MG[4].E_INCVar : INC-Variable / INC variable / Variable INC
   // // MG[5].E_INCVar : INC-Variable / INC variable / Variable INC
   // // MG[6].E_INCVar : INC-Variable / INC variable / Variable INC
   // // MG[7].E_INCVar : INC-Variable / INC variable / Variable INC
   // // MG[8].E_INCVar : INC-Variable / INC variable / Variable INC
   // // MG[9].E_INCVar : INC-Variable / INC variable / Variable INC
   // // MG[10].E_INCVar : INC-Variable / INC variable / Variable INC
   // // MG[3].E_ContManTravelAct : Kontinuierliches manuelles Verfahren aktiv / Continuous manual travel active / Desplazamiento manual continuo activo
   // // MG[4].E_ContManTravelAct : Kontinuierliches manuelles Verfahren aktiv / Continuous manual travel active / Desplazamiento manual continuo activo
   // // MG[5].E_ContManTravelAct : Kontinuierliches manuelles Verfahren aktiv / Continuous manual travel active / Desplazamiento manual continuo activo
   // // MG[6].E_ContManTravelAct : Kontinuierliches manuelles Verfahren aktiv / Continuous manual travel active / Desplazamiento manual continuo activo
   // // MG[7].E_ContManTravelAct : Kontinuierliches manuelles Verfahren aktiv / Continuous manual travel active / Desplazamiento manual continuo activo
   // // MG[8].E_ContManTravelAct : Kontinuierliches manuelles Verfahren aktiv / Continuous manual travel active / Desplazamiento manual continuo activo
   // // MG[9].E_ContManTravelAct : Kontinuierliches manuelles Verfahren aktiv / Continuous manual travel active / Desplazamiento manual continuo activo
   // // MG[10].E_ContManTravelAct : Kontinuierliches manuelles Verfahren aktiv / Continuous manual travel active / Desplazamiento manual continuo activo
   // // MG[3].E_HMI_INC1 : INC1 vom HMI / INC1 from HMI / INC1 de HMI
   // // MG[4].E_HMI_INC1 : INC1 vom HMI / INC1 from HMI / INC1 de HMI
   // // MG[5].E_HMI_INC1 : INC1 vom HMI / INC1 from HMI / INC1 de HMI
   // // MG[6].E_HMI_INC1 : INC1 vom HMI / INC1 from HMI / INC1 de HMI
   // // MG[7].E_HMI_INC1 : INC1 vom HMI / INC1 from HMI / INC1 de HMI
   // // MG[8].E_HMI_INC1 : INC1 vom HMI / INC1 from HMI / INC1 de HMI
   // // MG[9].E_HMI_INC1 : INC1 vom HMI / INC1 from HMI / INC1 de HMI
   // // MG[10].E_HMI_INC1 : INC1 vom HMI / INC1 from HMI / INC1 de HMI
   // // MG[3].E_HMI_INC10 : INC10 vom HMI / INC10 from HMI / INC10 de HMI
   // // MG[4].E_HMI_INC10 : INC10 vom HMI / INC10 from HMI / INC10 de HMI
   // // MG[5].E_HMI_INC10 : INC10 vom HMI / INC10 from HMI / INC10 de HMI
   // // MG[6].E_HMI_INC10 : INC10 vom HMI / INC10 from HMI / INC10 de HMI
   // // MG[7].E_HMI_INC10 : INC10 vom HMI / INC10 from HMI / INC10 de HMI
   // // MG[8].E_HMI_INC10 : INC10 vom HMI / INC10 from HMI / INC10 de HMI
   // // MG[9].E_HMI_INC10 : INC10 vom HMI / INC10 from HMI / INC10 de HMI
   // // MG[10].E_HMI_INC10 : INC10 vom HMI / INC10 from HMI / INC10 de HMI
   // // MG[3].E_HMI_INC100 : INC100 vom HMI / INC100 from HMI / INC100 de HMI
   // // MG[4].E_HMI_INC100 : INC100 vom HMI / INC100 from HMI / INC100 de HMI
   // // MG[5].E_HMI_INC100 : INC100 vom HMI / INC100 from HMI / INC100 de HMI
   // // MG[6].E_HMI_INC100 : INC100 vom HMI / INC100 from HMI / INC100 de HMI
   // // MG[7].E_HMI_INC100 : INC100 vom HMI / INC100 from HMI / INC100 de HMI
   // // MG[8].E_HMI_INC100 : INC100 vom HMI / INC100 from HMI / INC100 de HMI
   // // MG[9].E_HMI_INC100 : INC100 vom HMI / INC100 from HMI / INC100 de HMI
   // // MG[10].E_HMI_INC100 : INC100 vom HMI / INC100 from HMI / INC100 de HMI
   // // MG[3].E_HMI_INC1000 : INC1000 vom HMI / INC1000 from HMI / INC1000 de HMI
   // // MG[4].E_HMI_INC1000 : INC1000 vom HMI / INC1000 from HMI / INC1000 de HMI
   // // MG[5].E_HMI_INC1000 : INC1000 vom HMI / INC1000 from HMI / INC1000 de HMI
   // // MG[6].E_HMI_INC1000 : INC1000 vom HMI / INC1000 from HMI / INC1000 de HMI
   // // MG[7].E_HMI_INC1000 : INC1000 vom HMI / INC1000 from HMI / INC1000 de HMI
   // // MG[8].E_HMI_INC1000 : INC1000 vom HMI / INC1000 from HMI / INC1000 de HMI
   // // MG[9].E_HMI_INC1000 : INC1000 vom HMI / INC1000 from HMI / INC1000 de HMI
   // // MG[10].E_HMI_INC1000 : INC1000 vom HMI / INC1000 from HMI / INC1000 de HMI
   // // MG[3].E_HMI_INC10000 : INC10000 vom HMI / INC10000 from HMI / INC10000 de HMI
   // // MG[4].E_HMI_INC10000 : INC10000 vom HMI / INC10000 from HMI / INC10000 de HMI
   // // MG[5].E_HMI_INC10000 : INC10000 vom HMI / INC10000 from HMI / INC10000 de HMI
   // // MG[6].E_HMI_INC10000 : INC10000 vom HMI / INC10000 from HMI / INC10000 de HMI
   // // MG[7].E_HMI_INC10000 : INC10000 vom HMI / INC10000 from HMI / INC10000 de HMI
   // // MG[8].E_HMI_INC10000 : INC10000 vom HMI / INC10000 from HMI / INC10000 de HMI
   // // MG[9].E_HMI_INC10000 : INC10000 vom HMI / INC10000 from HMI / INC10000 de HMI
   // // MG[10].E_HMI_INC10000 : INC10000 vom HMI / INC10000 from HMI / INC10000 de HMI
   // // MG[3].E_HMI_INCVar : INC-Variable vom HMI / INC variable from HMI / Variable INC de HMI
   // // MG[4].E_HMI_INCVar : INC-Variable vom HMI / INC variable from HMI / Variable INC de HMI
   // // MG[5].E_HMI_INCVar : INC-Variable vom HMI / INC variable from HMI / Variable INC de HMI
   // // MG[6].E_HMI_INCVar : INC-Variable vom HMI / INC variable from HMI / Variable INC de HMI
   // // MG[7].E_HMI_INCVar : INC-Variable vom HMI / INC variable from HMI / Variable INC de HMI
   // // MG[8].E_HMI_INCVar : INC-Variable vom HMI / INC variable from HMI / Variable INC de HMI
   // // MG[9].E_HMI_INCVar : INC-Variable vom HMI / INC variable from HMI / Variable INC de HMI
   // // MG[10].E_HMI_INCVar : INC-Variable vom HMI / INC variable from HMI / Variable INC de HMI
   // // MG[3].E_HMI_ContManTravel : Kontinuierliches manuelles Verfahren vom HMI aktiv / Continuous manual travel active from HMI / Desplazamiento manual continuo activo desde HMI
   // // MG[4].E_HMI_ContManTravel : Kontinuierliches manuelles Verfahren vom HMI aktiv / Continuous manual travel active from HMI / Desplazamiento manual continuo activo desde HMI
   // // MG[5].E_HMI_ContManTravel : Kontinuierliches manuelles Verfahren vom HMI aktiv / Continuous manual travel active from HMI / Desplazamiento manual continuo activo desde HMI
   // // MG[6].E_HMI_ContManTravel : Kontinuierliches manuelles Verfahren vom HMI aktiv / Continuous manual travel active from HMI / Desplazamiento manual continuo activo desde HMI
   // // MG[7].E_HMI_ContManTravel : Kontinuierliches manuelles Verfahren vom HMI aktiv / Continuous manual travel active from HMI / Desplazamiento manual continuo activo desde HMI
   // // MG[8].E_HMI_ContManTravel : Kontinuierliches manuelles Verfahren vom HMI aktiv / Continuous manual travel active from HMI / Desplazamiento manual continuo activo desde HMI
   // // MG[9].E_HMI_ContManTravel : Kontinuierliches manuelles Verfahren vom HMI aktiv / Continuous manual travel active from HMI / Desplazamiento manual continuo activo desde HMI
   // // MG[10].E_HMI_ContManTravel : Kontinuierliches manuelles Verfahren vom HMI aktiv / Continuous manual travel active from HMI / Desplazamiento manual continuo activo desde HMI
   // // MG[2] : Nächste Betriebsartengruppe vom DBB20, wie bisher / next mode group from DBB20, as before / Próximo grupo de modos de operación del DBB20 como hasta ahora
   // // MG[3] : Nächste Betriebsartengruppe vom DBB20, wie bisher / next mode group from DBB20, as before / Próximo grupo de modos de operación del DBB20 como hasta ahora
   // // MG[4] : Nächste Betriebsartengruppe vom DBB20, wie bisher / next mode group from DBB20, as before / Próximo grupo de modos de operación del DBB20 como hasta ahora
   // // MG[5] : Nächste Betriebsartengruppe vom DBB20, wie bisher / next mode group from DBB20, as before / Próximo grupo de modos de operación del DBB20 como hasta ahora
   // // MG[6] : Nächste Betriebsartengruppe vom DBB20, wie bisher / next mode group from DBB20, as before / Próximo grupo de modos de operación del DBB20 como hasta ahora
   // // MG[7] : Nächste Betriebsartengruppe vom DBB20, wie bisher / next mode group from DBB20, as before / Próximo grupo de modos de operación del DBB20 como hasta ahora
   // // MG[8] : Nächste Betriebsartengruppe vom DBB20, wie bisher / next mode group from DBB20, as before / Próximo grupo de modos de operación del DBB20 como hasta ahora
   // // MG[9] : Nächste Betriebsartengruppe vom DBB20, wie bisher / next mode group from DBB20, as before / Próximo grupo de modos de operación del DBB20 como hasta ahora
   // // MG[10] : Nächste Betriebsartengruppe vom DBB20, wie bisher / next mode group from DBB20, as before / Próximo grupo de modos de operación del DBB20 como hasta ahora
END_TYPE

